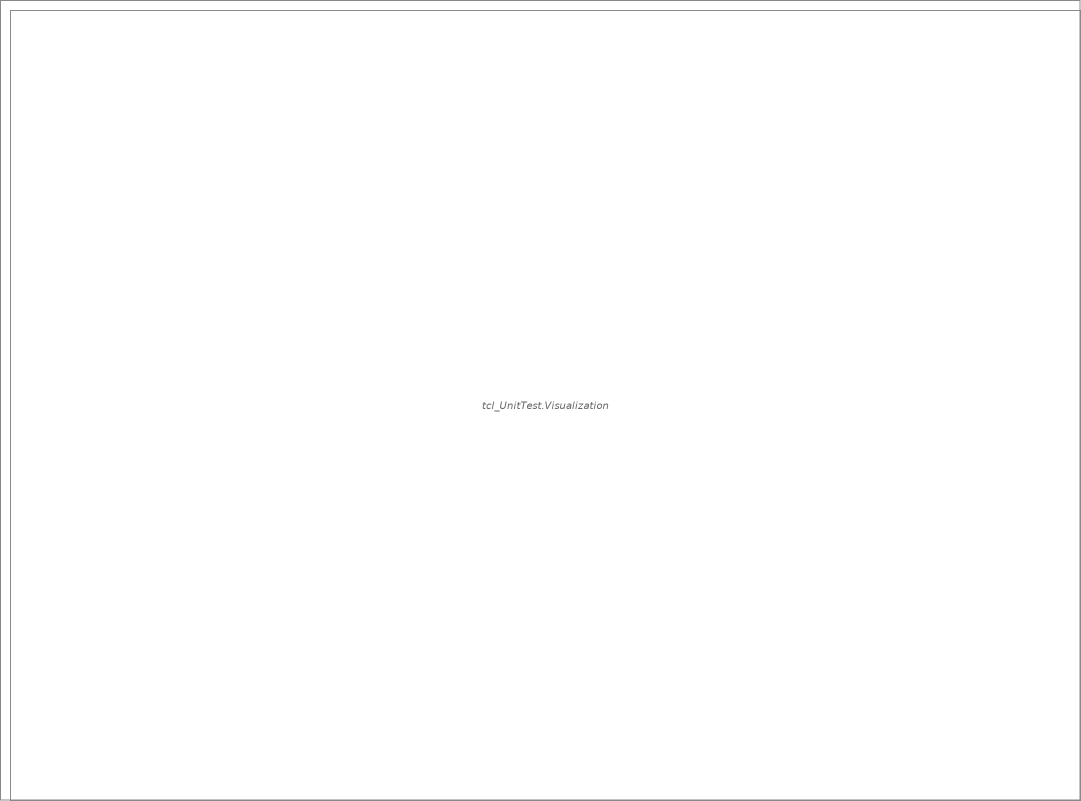
VISUALIZATION Visualization  // 1081x801
    Frame (10,10 1071x791)
        shows tcl_UnitTest.Visualization()
END_VISUALIZATION

(* stored: Version 1.1.0.1, ProductVersion 3.1.4024.3
   Visu Visualization: Id {b82bce25-4c01-0760-04b0-40b7e64cc1d3} *)
